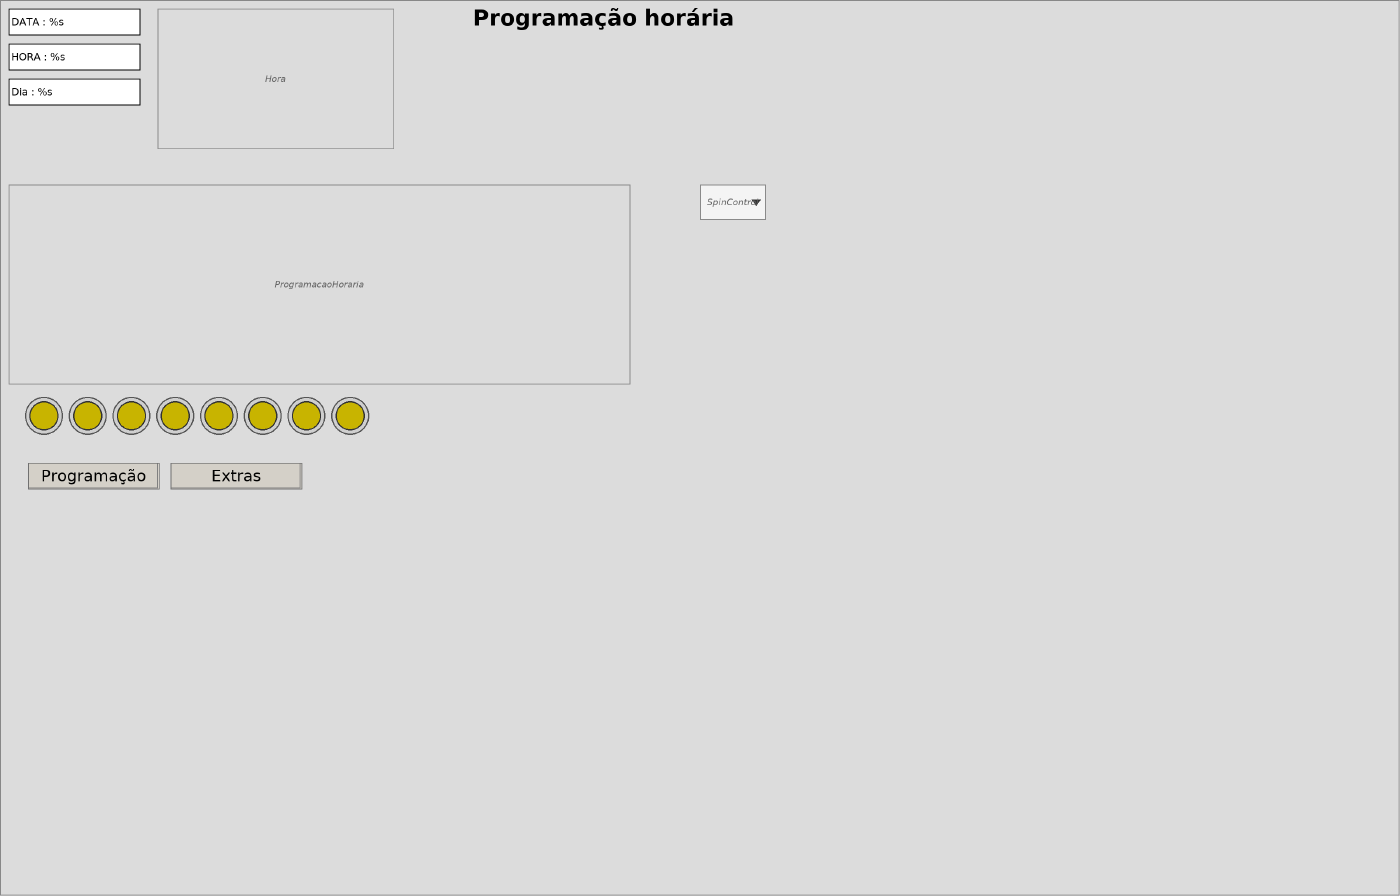
VISUALIZATION Visualization  // 1600x1024
    Rectangle (10,10 150x30), "DATA : %s", text variable: GVL_TimeSch.sActualDate
    Rectangle (10,50 150x30), "HORA : %s", text variable: GVL_TimeSch.sActualTime
    TabControl (180,10 270x160)
        shows Hora()
        shows Data()
        [0]: TabTitle=Acertar Hora
        [1]: TabTitle=Acertar Data
    TabControl (10,211 710x228)
        shows ProgramacaoHoraria(uiIndex := GVL_TimeSch.uiIndexToCheck, wDayOfWeek := GVL_TimeSch.ciMonday)
        shows ProgramacaoHoraria(uiIndex := GVL_TimeSch.uiIndexToCheck, wDayOfWeek := GVL_TimeSch.ciTuesday)
        shows ProgramacaoHoraria(uiIndex := GVL_TimeSch.uiIndexToCheck, wDayOfWeek := GVL_TimeSch.ciWednesday)
        shows ProgramacaoHoraria(uiIndex := GVL_TimeSch.uiIndexToCheck, wDayOfWeek := GVL_TimeSch.ciThursday)
        shows ProgramacaoHoraria(uiIndex := GVL_TimeSch.uiIndexToCheck, wDayOfWeek := GVL_TimeSch.ciFriday)
        shows ProgramacaoHoraria(uiIndex := GVL_TimeSch.uiIndexToCheck, wDayOfWeek := GVL_TimeSch.ciSaturday)
        shows ProgramacaoHoraria(uiIndex := GVL_TimeSch.uiIndexToCheck, wDayOfWeek := GVL_TimeSch.ciSunday)
        [0]: TabTitle=Segunda
        [1]: TabTitle=Terça
        [2]: TabTitle=Quarta
        [3]: TabTitle=Quinta
        [4]: TabTitle=Sexta
        [5]: TabTitle=Sabado
        [6]: TabTitle=Domingo
    Rectangle (10,90 150x30), "Dia : %s", text variable: GVL_TimeSch.sWeekDay
    SpinControl (800,211 75x40), variable: GVL_TimeSch.uiIndexToCheck
        p651134158: GVL_TimeSch.cNumberOfEventSchedules
    Group (25,450 400x50)
        Lamp1 (0,0 50x50), variable: GVL_TimeSch.abOutScheduler[1], style: Lamp-Lamp1-Yellow
        Lamp1 (50,0 50x50), variable: GVL_TimeSch.abOutScheduler[2], style: Lamp-Lamp1-Yellow
        Lamp1 (100,0 50x50), variable: GVL_TimeSch.abOutScheduler[3], style: Lamp-Lamp1-Yellow
        Lamp1 (150,0 50x50), variable: GVL_TimeSch.abOutScheduler[4], style: Lamp-Lamp1-Yellow
        Lamp1 (200,0 50x50), variable: GVL_TimeSch.abOutScheduler[5], style: Lamp-Lamp1-Yellow
        Lamp1 (250,0 50x50), variable: GVL_TimeSch.abOutScheduler[6], style: Lamp-Lamp1-Yellow
        Lamp1 (300,0 50x50), variable: GVL_TimeSch.abOutScheduler[7], style: Lamp-Lamp1-Yellow
        Lamp1 (350,0 50x50), variable: GVL_TimeSch.abOutScheduler[8], style: Lamp-Lamp1-Yellow
    Label (500,5 380x30), "Programação horária"
    Button (32,529 150x30), "Programação"
        OnMouseClick: change screen: Visualization
    Button (195,529 150x30), "Extras"
        OnMouseClick: change screen: FuncoesExtras
END_VISUALIZATION

(* stored: Version 1.1.0.1, ProductVersion 3.1.4024.11
   Visu Visualization: Id {83ad0cab-e56b-4a6c-822c-8ce441948034} *)
